FUNCTION_BLOCK FB_SVs_Output
VAR_INPUT
	Stellung : BOOL;
END_VAR
VAR_OUTPUT
	OUT_Stellung : BOOL;
END_VAR
VAR
END_VAR

OUT_Stellung := Stellung;

END_FUNCTION_BLOCK

(* stored: Version 1.1.0.1, ProductVersion 3.1.4024.9
   POU FB_SVs_Output: Id {0c8b6cec-f274-4b5d-b0c7-cf08d41ebbf8}, SpecialFunc None *)
